// TIA Portal V19 export
TYPE "typeU2Em4Para"
// stored: Access Published
   STRUCT
      cm1SV112 : "typeAxisControlInterface";
      cm2SV113 { S7_SetPoint := 'True'} : "typeAxisControlInterface";
      cm3SV115 { S7_SetPoint := 'True'} : "typeAxisControlInterface";
      cm4SV116 { S7_SetPoint := 'True'} : "typeAxisControlInterface";
   END_STRUCT;
END_TYPE
